TYPE ST_BigBagChangeHandlerOutValues :
STRUCT
	    rBagInitialMass 	 : REAL; // masa początkowa aktualnie założonego worka zadana przez operatora ze SCADA
END_STRUCT
END_TYPE

(* stored: Version 1.1.0.1, ProductVersion 3.1.4024.16
   DUT ST_BigBagChangeHandlerOutValues: Id {f115d36f-8cc8-47c2-a564-390b08c33571} *)
